INTERFACE ITF_Actuator

METHOD Advance
VAR_INPUT
END_VAR
END_METHOD

PROPERTY P_Advanced : BOOL
GET
END_GET
END_PROPERTY

PROPERTY P_OperatorControl : BOOL
GET
END_GET
SET
END_SET
END_PROPERTY

PROPERTY P_OperatorValue : E_State
GET
END_GET
SET
END_SET
END_PROPERTY

PROPERTY P_Retracted : BOOL
GET
END_GET
END_PROPERTY

METHOD Retract
VAR_INPUT
END_VAR
END_METHOD

END_INTERFACE

(* stored: Version 1.1.0.1
   Itf ITF_Actuator: Id {d20148bd-fb54-4987-a2f5-6ed5b6f075de}
   Folder Methods: Id {7e00d6e6-8714-414d-86fb-f3a31f687736}
   Folder Properties: Id {0f9b9193-2187-4ab0-aee6-f55532e80ee4}
   Method Advance: Id {e1872d33-0934-40fc-abcc-5017c8e66648}
   Property P_Advanced: Id {60cf6693-3f78-4700-9cd6-17e9a60c3593}
   Get Get: Id {660e5fe7-4dff-47b0-a908-e3f8c27e919c}
   Property P_OperatorControl: Id {2fb28d7f-2749-44b8-992b-9e5915adc993}
   Get Get: Id {c3a5eeea-7f03-443e-9473-12d316facb0e}
   Set Set: Id {3c48ec13-f4bc-4732-a747-381ac5966439}
   Property P_OperatorValue: Id {9b95ce3b-e9c4-4417-8ca0-76c05f4fa5d2}
   Get Get: Id {f0dcbe40-bfbc-4aa2-8ad0-add79c12e432}
   Set Set: Id {1c725391-c913-4d99-ac8b-96f837fd61b4}
   Property P_Retracted: Id {609d519f-1d8c-4864-bd7d-50c6f28153fc}
   Get Get: Id {d2ac7f15-dbe8-4a6f-9446-24003236a7cd}
   Method Retract: Id {cb0ee7f0-3202-4ce7-907c-31b917761528} *)
